VAR_GLOBAL
	Module		: ARRAY [1..GrpCnt] OF DUT_MODULE_INTERFACE;
	
END_VAR

(* stored: Version 1.1.0.1, ProductVersion 3.1.0.25
   GVL ModuleInterface: Id {d214e4e1-e1cc-4d4d-9969-055a64012ea6} *)
